// Mitsubishi GX Works2 project: Group1 extracted   PLC: FX3U/FX3UC

PROGRAM MAIN
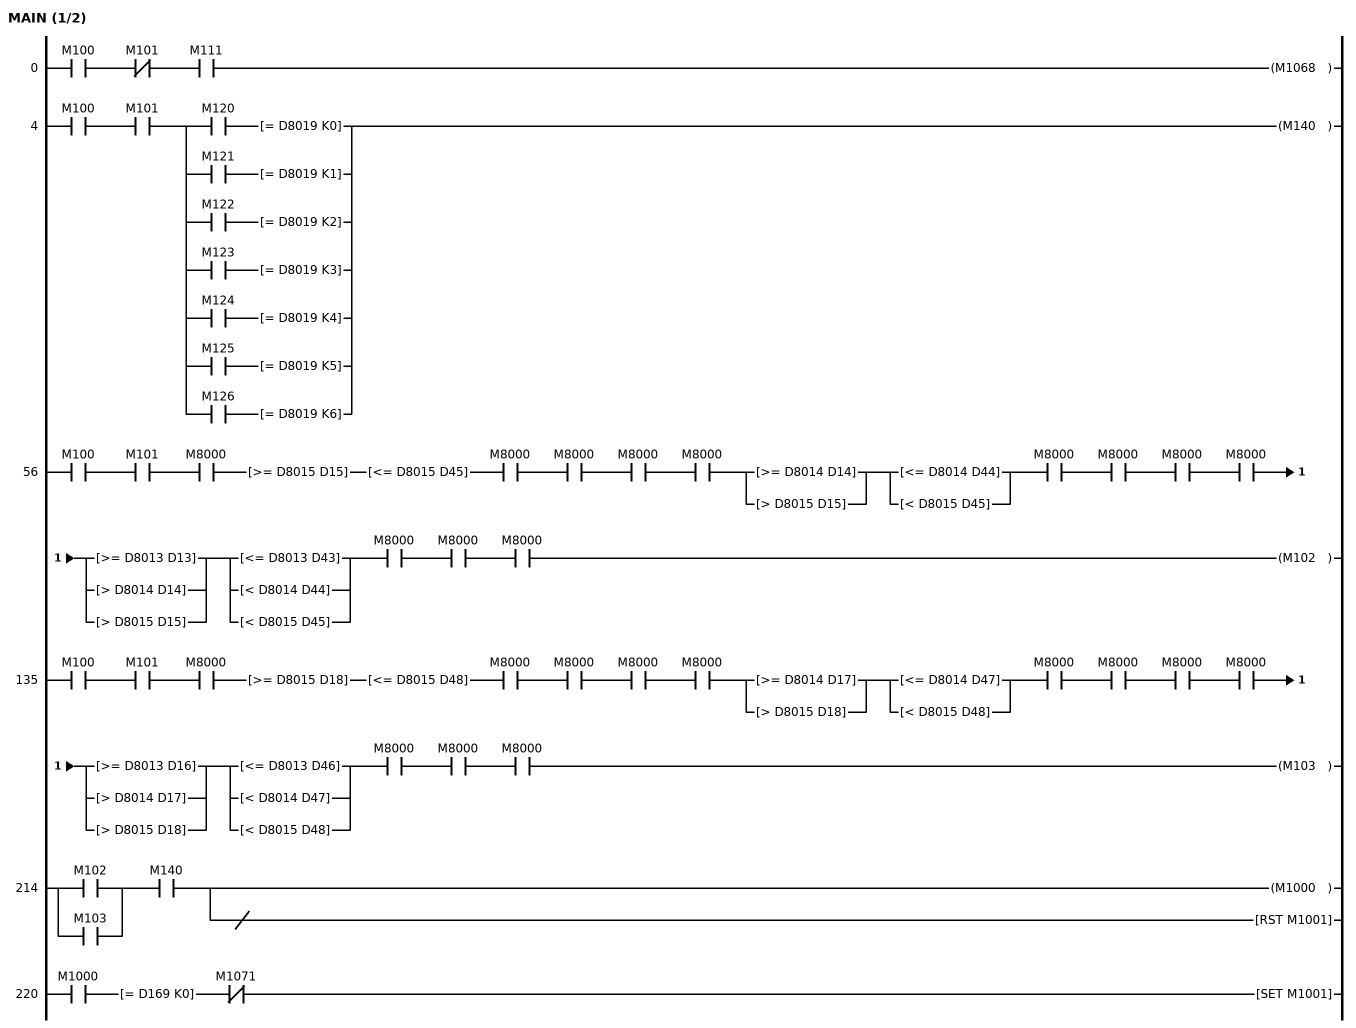
0     LD      M100
      ANI     M101
      AND     M111
      OUT     M1068
4     LD      M100
      AND     M101
      LD      M120
      AND=    D8019 K0
      LD      M121
      AND=    D8019 K1
      ORB
      LD      M122
      AND=    D8019 K2
      ORB
      LD      M123
      AND=    D8019 K3
      ORB
      LD      M124
      AND=    D8019 K4
      ORB
      LD      M125
      AND=    D8019 K5
      ORB
      LD      M126
      AND=    D8019 K6
      ORB
      ANB
      OUT     M140
56    LD      M100
      AND     M101
      AND     M8000
      AND>=   D8015 D15
      AND<=   D8015 D45
      AND     M8000
      AND     M8000
      AND     M8000
      AND     M8000
      LD>=    D8014 D14
      OR>     D8015 D15
      ANB
      LD<=    D8014 D44
      OR<     D8015 D45
      ANB
      AND     M8000
      AND     M8000
      AND     M8000
      AND     M8000
      LD>=    D8013 D13
      OR>     D8014 D14
      OR>     D8015 D15
      ANB
      LD<=    D8013 D43
      OR<     D8014 D44
      OR<     D8015 D45
      ANB
      AND     M8000
      AND     M8000
      AND     M8000
      OUT     M102
135   LD      M100
      AND     M101
      AND     M8000
      AND>=   D8015 D18
      AND<=   D8015 D48
      AND     M8000
      AND     M8000
      AND     M8000
      AND     M8000
      LD>=    D8014 D17
      OR>     D8015 D18
      ANB
      LD<=    D8014 D47
      OR<     D8015 D48
      ANB
      AND     M8000
      AND     M8000
      AND     M8000
      AND     M8000
      LD>=    D8013 D16
      OR>     D8014 D17
      OR>     D8015 D18
      ANB
      LD<=    D8013 D46
      OR<     D8014 D47
      OR<     D8015 D48
      ANB
      AND     M8000
      AND     M8000
      AND     M8000
      OUT     M103
214   LD      M102
      OR      M103
      AND     M140
      OUT     M1000
      INV
      RST     M1001
220   LD      M1000
      AND=    D169 K0
      ANI     M1071
      SET     M1001
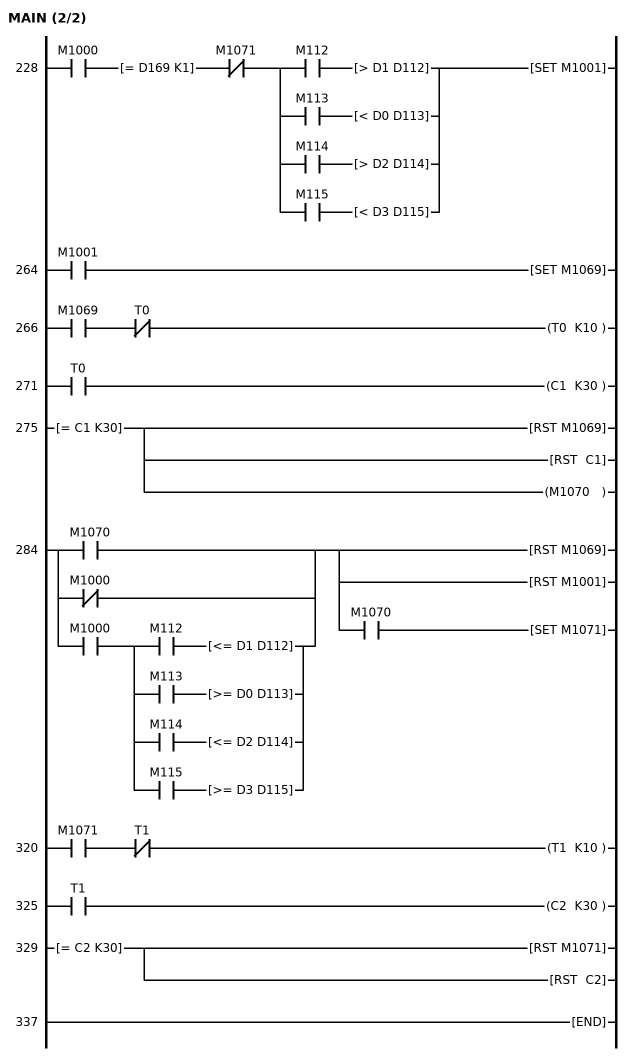
228   LD      M1000
      AND=    D169 K1
      ANI     M1071
      LD      M112
      AND>    D1 D112
      LD      M113
      AND<    D0 D113
      ORB
      LD      M114
      AND>    D2 D114
      ORB
      LD      M115
      AND<    D3 D115
      ORB
      ANB
      SET     M1001
264   LD      M1001
      SET     M1069
266   LD      M1069
      ANI     T0
      OUT     T0 K10
271   LD      T0
      OUT     C1 K30
275   LD=     C1 K30
      RST     M1069
      RST     C1
      OUT     M1070
284   LD      M1070
      ORI     M1000
      LD      M1000
      LD      M112
      AND<=   D1 D112
      LD      M113
      AND>=   D0 D113
      ORB
      LD      M114
      AND<=   D2 D114
      ORB
      LD      M115
      AND>=   D3 D115
      ORB
      ANB
      ORB
      RST     M1069
      RST     M1001
      AND     M1070
      SET     M1071
320   LD      M1071
      ANI     T1
      OUT     T1 K10
325   LD      T1
      OUT     C2 K30
329   LD=     C2 K30
      RST     M1071
      RST     C2
337   END
END_PROGRAM
